// TIA Portal V21 export
VAR_GLOBAL   // PLC tag table "K_TipoOutValvola"
END_VAR
VAR_GLOBAL CONSTANT   // user constants
   K_TipoOutValvola_Portata : Int := 1;
   K_TipoOutValvola_Pressione : Int := 2;
END_VAR
